(*
Searches an `I_Entity` for a `I_Tag` component matching provided id pattern.
Result:
- Ok - Returns iTag.
- Err.NotFound - Returns null.
- Err.InvRef - Provided reference is invalid.
- Err.Itf0 - Returns null, incorrect interface.
*)
FUNCTION GetTag : Result
VAR_INPUT
	iEntity		: I_Entity;
	sIdPattern	: Str;
	iOut		: REFERENCE TO I_Tag;
END_VAR
VAR
	_iComp		: I_Component;
	cmp			: TagCmp;
END_VAR

IF iEntity = 0 THEN
	GetTag := Err.Itf0;
	RETURN;
END_IF

IF NOT __ISVALIDREF(iOut) THEN
	GetTag := Err.InvRef;
	RETURN;
END_IF

WHILE IsOk(iEntity.GetNextComp(_iComp)) DO
	IF IsOk(ICompToITag(_iComp.Raw, iOut)) THEN
		IF cmp.Set(iOut).MatchWcdId(sIdPattern).IsTrue() THEN
			GetTag := Ok;
			RETURN;
		ELSE
			iOut := 0;
		END_IF
	END_IF
END_WHILE

GetTag := Err.NotFound;

END_FUNCTION

(* stored: Version 1.1.0.1
   POU GetTag: Id {99d2f861-a98d-4a03-974c-921613e65770}, SpecialFunc None *)
